Xinje XDPPro project, PLC1: XD3-16 (software 3.7.17b 2023-10-13)

PROGRAM Ladder

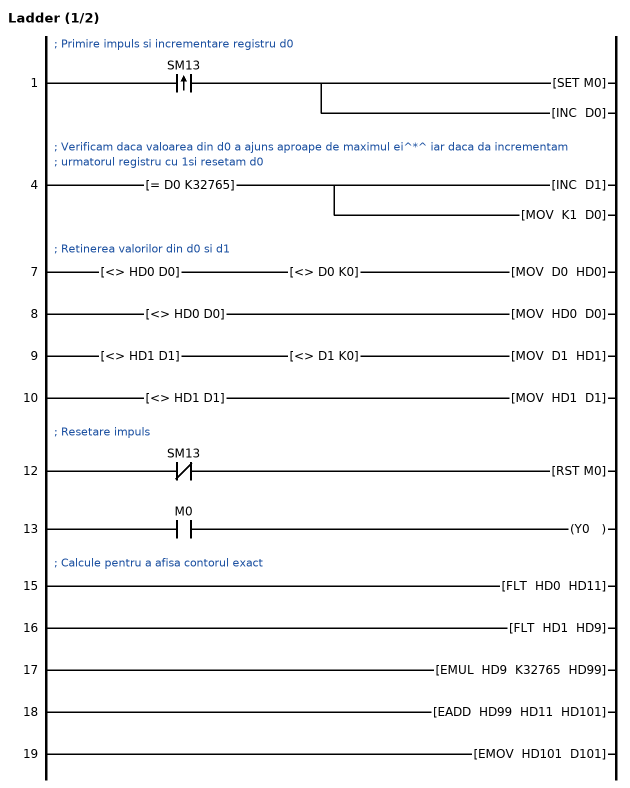
; Primire impuls si incrementare registru d0
LDP    SM13
SET    M0
INC    D0
; Verificam daca valoarea din d0 a ajuns aproape de maximul ei^*^ iar daca da incrementam urmatorul registru cu 1si resetam d0
LD=    D0 K32765
INC    D1
MOV    K1 D0
; Retinerea valorilor din d0 si d1
LD<>   HD0 D0
AND<>  D0 K0
MOV    D0 HD0
LD<>   HD0 D0
MOV    HD0 D0
LD<>   HD1 D1
AND<>  D1 K0
MOV    D1 HD1
LD<>   HD1 D1
MOV    HD1 D1
; Resetare impuls
LDI    SM13
RST    M0
LD     M0
OUT    Y0
; Calcule pentru a afisa contorul exact
FLT    HD0 HD11
FLT    HD1 HD9
EMUL   HD9 K32765 HD99
EADD   HD99 HD11 HD101
EMOV   HD101 D101

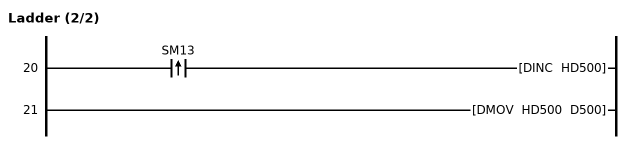
LDP    SM13
DINC   HD500
DMOV   HD500 D500